// TIA Portal V19 export
VAR_GLOBAL   // PLC tag table "D05"
   D05_Lp_EntryReq_LB122 AT %Q107.3 : Bool;   // 193SH1
   D05_Lp_SafetyReset_LB122 AT %Q107.4 : Bool;   // 193SH2
   D05_Pb_EntryReq_LB122 AT %I104.0 : Bool;   // 193SH1
   D05_Pb_SafetyReset_LB122 AT %I104.1 : Bool;   // 193SH2
   D05_Unlock AT %Q107.2 : Bool;   // 19302 Comando elettroserratura
   D05_LockEnable AT %I103.6 : Bool;   // 19301 Cancello chiuso
   D05_Cancello_Bloccato AT %I103.7 : Bool;   // 19303
   D05_Ls AT %I1027.0 : Bool;   // 103DI0 - 193A1
END_VAR
